// TIA Portal V18 export
FUNCTION "ST10_Tip" : Void   // FC1007, LAD
{ S7_Optimized_Access := 'FALSE' }
VERSION : 0.1
// stored: AutoNumber false, IsIECCheckEnabled false, SetENOAutomatically false, UDAEnableTagReadback false
   VAR_TEMP   // added for the SCL form of the ladder/FBD networks
      _w1 : Bool;
   END_VAR
BEGIN

NETWORK
TITLE = Gloal Tips

//7000: 设备未上电，请先按下复位按钮，在按下控制开按钮
//      AN    "iHMIE-StopPB"
//     AN    "iE_StopPB_1"
//     AN    "iE_StopPB_2"
//     AN    "iE_StopPB_3"
//     AN    "ST350_Sys".Status.ControlOn
//     =     "ST350_TipDB".Global."1".ControlOn

//7001：设备存在故障，请查看报警信息，消除故障，然后按复位按钮
//     A     "ST350_Sys".Status.ControlOn
//     O(
//      A     "iHMIE-StopPB"
//     O     "iE_StopPB_1"
//     O     "iE_StopPB_2"
//     O     "iE_StopPB_3"
//    )
//    A     "ST350_Sys".Alarm.ON
//    =     "ST350_TipDB".Global."1".Reset

//7002: 未选择配方，请在换型页面选择配方
//      A     "ST350_Sys".Status.ControlOn
//     AN    "ST350_TipDB".Global."1".Reset
//
//      AN    "ST350_RecipeDB".Recipe.Equal
//     =     "ST350_TipDB".Global."2"[0]

//7003:设备未选择自动，请选择自动模式
//      A     "ST350_Sys".Status.ControlOn
//     AN    "ST350_TipDB".Global."1".Reset
//     A     "ST350_RecipeDB".Recipe.Equal
//     AN    "ST350_Sys".Interface.Auto.Mode

//    =     "ST350_TipDB".Global."1".SelectAutoMode

//7004:设备初始化，请启动设备初始化
//     A     "ST350_Sys".Status.ControlOn
//     AN    "ST350_TipDB".Global."1".Reset
//      A     "ST350_RecipeDB".Recipe.Equal
//     A     "ST350_Sys".Interface.Auto.Mode

//    AN    "ST350_Sys".Initial.OK
//     =     "ST350_TipDB".Global."2"[1]


//7005:设备未启动，请启动自动运行
//     A     "ST350_Sys".Status.ControlOn
//    AN    "ST350_TipDB".Global."1".Reset
//    A     "ST350_RecipeDB".Recipe.Equal
//    A     "ST350_Sys".Interface.Auto.Mode
//    A     "ST350_Sys".Initial.OK
//
//    AN    "ST350_Sys".Interface.Auto.Running
//    AN    "ST350_Sys".Interface.Auto.AllRun
//    =     "ST350_TipDB".Global."1".AutoModeRunning

REGION Network 2: Gloal Tips:7000: 设备未上电，请先按下复位按钮，在按下控制开按钮 / Gloal Tips:7000: The device is not powered on, please press the reset button first, and then press the control button
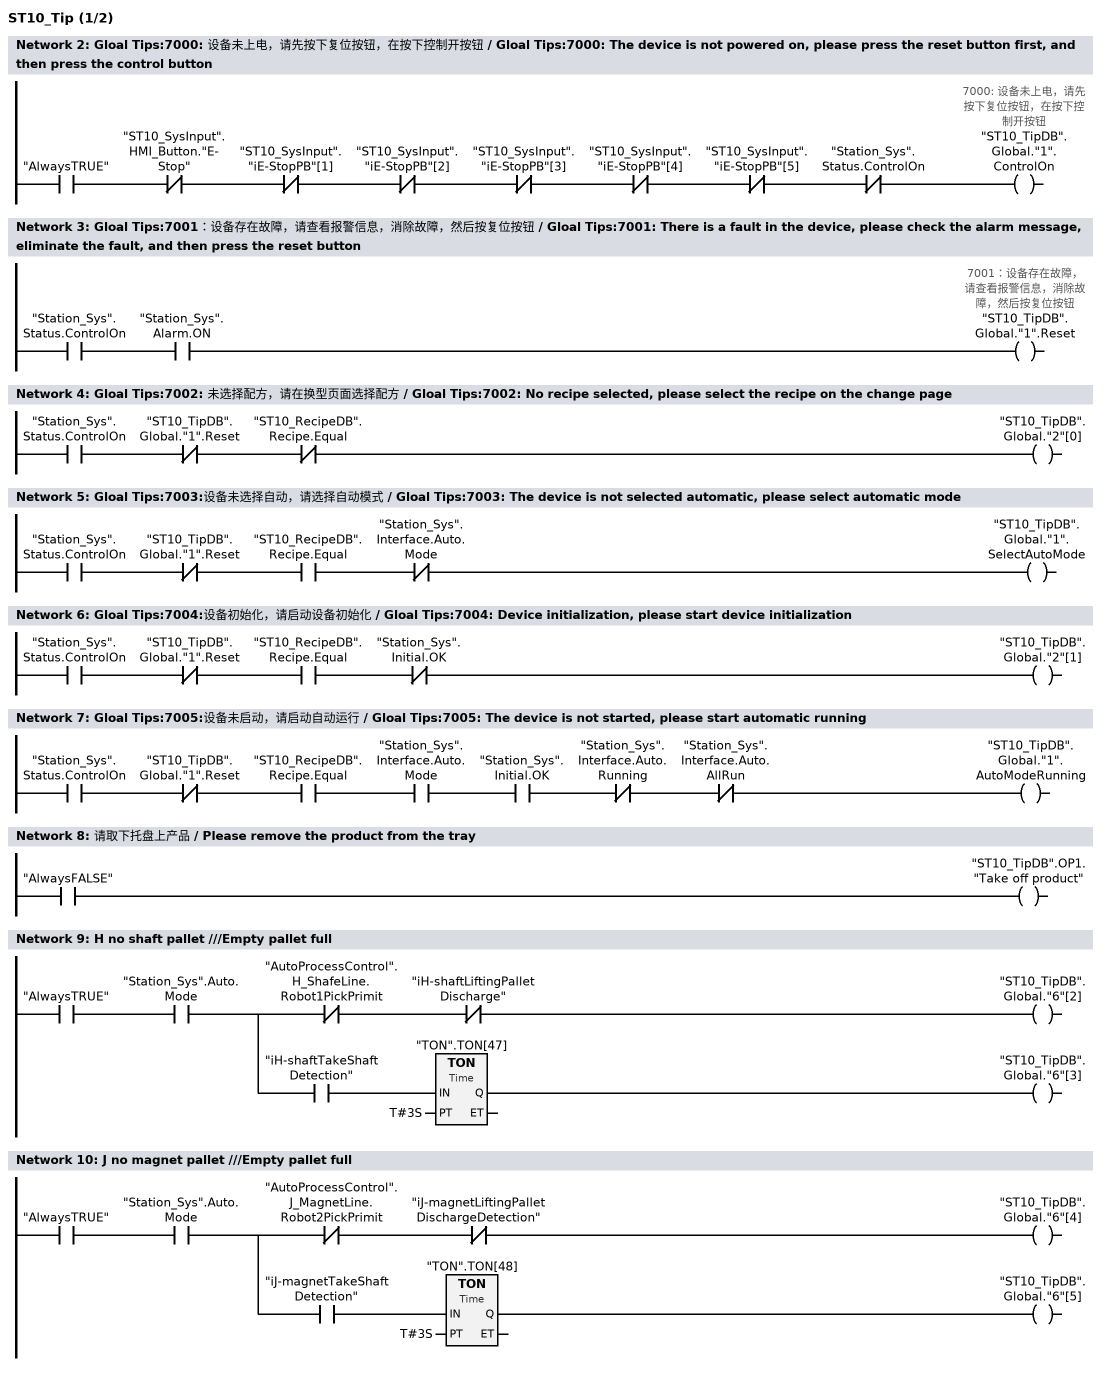
   RUNG wire#powerrail
      Contact( "AlwaysTRUE" )
      I_Contact( "ST10_SysInput".HMI_Button."E-Stop" )
      I_Contact( "ST10_SysInput"."iE-StopPB"[1] )
      I_Contact( "ST10_SysInput"."iE-StopPB"[2] )
      I_Contact( "ST10_SysInput"."iE-StopPB"[3] )
      I_Contact( "ST10_SysInput"."iE-StopPB"[4] )
      I_Contact( "ST10_SysInput"."iE-StopPB"[5] )
      I_Contact( "Station_Sys".Status.ControlOn )
      Coil( "ST10_TipDB".Global."1".ControlOn )   // 7000: 设备未上电，请先按下复位按钮，在按下控制开按钮
   END_RUNG
   // the same network as SCL:
   "ST10_TipDB".Global."1".ControlOn := "AlwaysTRUE" AND NOT "ST10_SysInput".HMI_Button."E-Stop" AND NOT "ST10_SysInput"."iE-StopPB"[1] AND NOT "ST10_SysInput"."iE-StopPB"[2] AND NOT "ST10_SysInput"."iE-StopPB"[3] AND NOT "ST10_SysInput"."iE-StopPB"[4] AND NOT "ST10_SysInput"."iE-StopPB"[5] AND NOT "Station_Sys".Status.ControlOn;   // 7000: 设备未上电，请先按下复位按钮，在按下控制开按钮
END_REGION

REGION Network 3: Gloal Tips:7001：设备存在故障，请查看报警信息，消除故障，然后按复位按钮 / Gloal Tips:7001: There is a fault in the device, please check the alarm message, eliminate the fault, and then press the reset button
   RUNG wire#powerrail
      Contact( "Station_Sys".Status.ControlOn )
      Contact( "Station_Sys".Alarm.ON )
      Coil( "ST10_TipDB".Global."1".Reset )   // 7001：设备存在故障，请查看报警信息，消除故障，然后按复位按钮
   END_RUNG
   // the same network as SCL:
   "ST10_TipDB".Global."1".Reset := "Station_Sys".Status.ControlOn AND "Station_Sys".Alarm.ON;   // 7001：设备存在故障，请查看报警信息，消除故障，然后按复位按钮
END_REGION

REGION Network 4: Gloal Tips:7002: 未选择配方，请在换型页面选择配方 / Gloal Tips:7002: No recipe selected, please select the recipe on the change page
   RUNG wire#powerrail
      Contact( "Station_Sys".Status.ControlOn )
      I_Contact( "ST10_TipDB".Global."1".Reset )
      I_Contact( "ST10_RecipeDB".Recipe.Equal )
      Coil( "ST10_TipDB".Global."2"[0] )
   END_RUNG
   // the same network as SCL:
   "ST10_TipDB".Global."2"[0] := "Station_Sys".Status.ControlOn AND NOT "ST10_TipDB".Global."1".Reset AND NOT "ST10_RecipeDB".Recipe.Equal;
END_REGION

REGION Network 5: Gloal Tips:7003:设备未选择自动，请选择自动模式 / Gloal Tips:7003: The device is not selected automatic, please select automatic mode
   RUNG wire#powerrail
      Contact( "Station_Sys".Status.ControlOn )
      I_Contact( "ST10_TipDB".Global."1".Reset )
      Contact( "ST10_RecipeDB".Recipe.Equal )
      I_Contact( "Station_Sys".Interface.Auto.Mode )
      Coil( "ST10_TipDB".Global."1".SelectAutoMode )
   END_RUNG
   // the same network as SCL:
   "ST10_TipDB".Global."1".SelectAutoMode := "Station_Sys".Status.ControlOn AND NOT "ST10_TipDB".Global."1".Reset AND "ST10_RecipeDB".Recipe.Equal AND NOT "Station_Sys".Interface.Auto.Mode;
END_REGION

REGION Network 6: Gloal Tips:7004:设备初始化，请启动设备初始化 / Gloal Tips:7004: Device initialization, please start device initialization
   RUNG wire#powerrail
      Contact( "Station_Sys".Status.ControlOn )
      I_Contact( "ST10_TipDB".Global."1".Reset )
      Contact( "ST10_RecipeDB".Recipe.Equal )
      I_Contact( "Station_Sys".Initial.OK )
      Coil( "ST10_TipDB".Global."2"[1] )
   END_RUNG
   // the same network as SCL:
   "ST10_TipDB".Global."2"[1] := "Station_Sys".Status.ControlOn AND NOT "ST10_TipDB".Global."1".Reset AND "ST10_RecipeDB".Recipe.Equal AND NOT "Station_Sys".Initial.OK;
END_REGION

REGION Network 7: Gloal Tips:7005:设备未启动，请启动自动运行 / Gloal Tips:7005: The device is not started, please start automatic running
   RUNG wire#powerrail
      Contact( "Station_Sys".Status.ControlOn )
      I_Contact( "ST10_TipDB".Global."1".Reset )
      Contact( "ST10_RecipeDB".Recipe.Equal )
      Contact( "Station_Sys".Interface.Auto.Mode )
      Contact( "Station_Sys".Initial.OK )
      I_Contact( "Station_Sys".Interface.Auto.Running )
      I_Contact( "Station_Sys".Interface.Auto.AllRun )
      Coil( "ST10_TipDB".Global."1".AutoModeRunning )
   END_RUNG
   // the same network as SCL:
   "ST10_TipDB".Global."1".AutoModeRunning := "Station_Sys".Status.ControlOn AND NOT "ST10_TipDB".Global."1".Reset AND "ST10_RecipeDB".Recipe.Equal AND "Station_Sys".Interface.Auto.Mode AND "Station_Sys".Initial.OK AND NOT "Station_Sys".Interface.Auto.Running AND NOT "Station_Sys".Interface.Auto.AllRun;
END_REGION

REGION Network 8: 请取下托盘上产品 / Please remove the product from the tray
   RUNG wire#powerrail
      Contact( "AlwaysFALSE" )
      Coil( "ST10_TipDB".OP1."Take off product" )
   END_RUNG
   // the same network as SCL:
   "ST10_TipDB".OP1."Take off product" := "AlwaysFALSE";
END_REGION

REGION Network 9: H no shaft pallet ///Empty pallet full
   RUNG wire#powerrail
      Contact( "AlwaysTRUE" )
      Contact( "Station_Sys".Auto.Mode )
      wire#w1
      I_Contact( "AutoProcessControl".H_ShafeLine.Robot1PickPrimit )
      I_Contact( "iH-shaftLiftingPalletDischarge" )
      Coil( "ST10_TipDB".Global."6"[2] )
   END_RUNG
   RUNG wire#w1
      Contact( "iH-shaftTakeShaftDetection" )
      { S7_Templates := "time_type := Time" } "TON".TON[47].TON(pt := T#3S, et =>)
      Coil( "ST10_TipDB".Global."6"[3] )
   END_RUNG
   // the same network as SCL:
   #_w1 := "AlwaysTRUE" AND "Station_Sys".Auto.Mode;
   "ST10_TipDB".Global."6"[2] := #_w1 AND NOT "AutoProcessControl".H_ShafeLine.Robot1PickPrimit AND NOT "iH-shaftLiftingPalletDischarge";
   "TON".TON[47].TON(IN := #_w1 AND "iH-shaftTakeShaftDetection", PT := T#3S);
   "ST10_TipDB".Global."6"[3] := "TON".TON[47].Q;
END_REGION

REGION Network 10: J no magnet pallet ///Empty pallet full
   RUNG wire#powerrail
      Contact( "AlwaysTRUE" )
      Contact( "Station_Sys".Auto.Mode )
      wire#w1
      I_Contact( "AutoProcessControl".J_MagnetLine.Robot2PickPrimit )
      I_Contact( "iJ-magnetLiftingPalletDischargeDetection" )
      Coil( "ST10_TipDB".Global."6"[4] )
   END_RUNG
   RUNG wire#w1
      Contact( "iJ-magnetTakeShaftDetection" )
      { S7_Templates := "time_type := Time" } "TON".TON[48].TON(pt := T#3S, et =>)
      Coil( "ST10_TipDB".Global."6"[5] )
   END_RUNG
   // the same network as SCL:
   #_w1 := "AlwaysTRUE" AND "Station_Sys".Auto.Mode;
   "ST10_TipDB".Global."6"[4] := #_w1 AND NOT "AutoProcessControl".J_MagnetLine.Robot2PickPrimit AND NOT "iJ-magnetLiftingPalletDischargeDetection";
   "TON".TON[48].TON(IN := #_w1 AND "iJ-magnetTakeShaftDetection", PT := T#3S);
   "ST10_TipDB".Global."6"[5] := "TON".TON[48].Q;
END_REGION

REGION Network 11: K no magnet pallet ///Empty pallet full
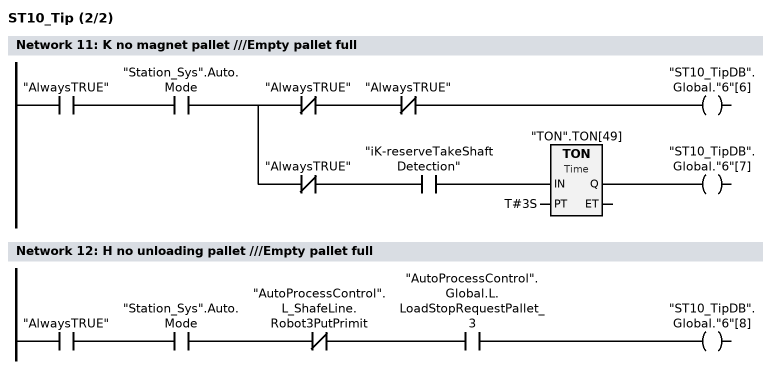
   RUNG wire#powerrail
      Contact( "AlwaysTRUE" )
      Contact( "Station_Sys".Auto.Mode )
      wire#w1
      I_Contact( "AlwaysTRUE" )
      I_Contact( "AlwaysTRUE" )
      Coil( "ST10_TipDB".Global."6"[6] )
   END_RUNG
   RUNG wire#w1
      I_Contact( "AlwaysTRUE" )
      Contact( "iK-reserveTakeShaftDetection" )
      { S7_Templates := "time_type := Time" } "TON".TON[49].TON(pt := T#3S, et =>)
      Coil( "ST10_TipDB".Global."6"[7] )
   END_RUNG
   // the same network as SCL:
   #_w1 := "AlwaysTRUE" AND "Station_Sys".Auto.Mode;
   "ST10_TipDB".Global."6"[6] := #_w1 AND NOT "AlwaysTRUE" AND NOT "AlwaysTRUE";
   "TON".TON[49].TON(IN := #_w1 AND NOT "AlwaysTRUE" AND "iK-reserveTakeShaftDetection", PT := T#3S);
   "ST10_TipDB".Global."6"[7] := "TON".TON[49].Q;
END_REGION

REGION Network 12: H no unloading pallet ///Empty pallet full
   RUNG wire#powerrail
      Contact( "AlwaysTRUE" )
      Contact( "Station_Sys".Auto.Mode )
      I_Contact( "AutoProcessControl".L_ShafeLine.Robot3PutPrimit )
      Contact( "AutoProcessControl".Global.L.LoadStopRequestPallet_3 )
      Coil( "ST10_TipDB".Global."6"[8] )
   END_RUNG
   // the same network as SCL:
   "ST10_TipDB".Global."6"[8] := "AlwaysTRUE" AND "Station_Sys".Auto.Mode AND NOT "AutoProcessControl".L_ShafeLine.Robot3PutPrimit AND "AutoProcessControl".Global.L.LoadStopRequestPallet_3;
END_REGION
END_FUNCTION
